# B&R Automation Studio project TD52 (part 8)

#### main.c
```c
/********************************************************************
 * COPYRIGHT -- Bernecker + Rainer Industrie-Elektronik Ges.m.b.H.
 ********************************************************************
 * Program: Sim3pCTR
 * File: main.c
 * Author: 105051472
 * Created: Thu Jan 10 08:03:20 2013
 ********************************************************************
 * Implementation of program Sim3pCTR
 ********************************************************************
 * Generated with B&R Automation Studio Target for Simulink V3.3
 * (ERT based)
 ********************************************************************/

#include <bur/plctypes.h>
#include "Sim3pCTR.h"
#include "rtwtypes.h"

BOOL bur_firsttime = TRUE;

/*  Defines */

/*  Data Types */

/**************************** GLOBAL DATA *************************************/
/*  Definitions */

/*  Declarations  */

/***************************** FILE SCOPE DATA ********************************/

/*************************** FUNCTIONS ****************************************/
#ifdef __cplusplus

unsigned long bur_heap_size = 65535;

#endif

void Sim3pCTR(struct Sim3pCTR* inst)
{
  switch (inst->ssMethodType)
  {
   case SS_INITIALIZE:
    /* call model initialize function */
    Sim3pCTR_initialize(inst);
    break;

   case SS_OUTPUT:
    /* call model step function */
    Sim3pCTR_step(inst);

    break;

   case SS_TERMINATE:
    /* call model terminate function */
    Sim3pCTR_terminate(inst);
    break;
  }
}

/*****************************************************************************
   Function block sample time: 0.01s
 *****************************************************************************/

/*****************************************************************************
   B&R Automation Studio Target for Simulink Version: V3.3.19 (13-Jun-2012)
 *****************************************************************************/

/*======================== TOOL VERSION INFORMATION ==========================*
 * MATLAB 7.12 (R2011a)09-Mar-2011                                            *
 * Simulink 7.7 (R2011a)09-Mar-2011                                           *
 * Simulink Coder 8.0 (R2011a)09-Mar-2011                                     *
 * Embedded Coder 6.0 (R2011a)09-Mar-2011                                     *
 * Stateflow 7.7 (R2011a)09-Mar-2011                                          *
 * Simulink Fixed Point 6.5 (R2011a)09-Mar-2011                               *
 *============================================================================*/

/*======================= LICENSE IN USE INFORMATION =========================*
 * matlab                                                                     *
 * matlab_coder                                                               *
 * real-time_workshop                                                         *
 * rtw_embedded_coder                                                         *
 * simulink                                                                   *
 * stateflow                                                                  *
 *============================================================================*/
```

#### lib_properties.txt
```
For manual assignment to hardware configuration please
add the following additional include directories:

\Logical\MATLAB_includes\R2011a\

And the following additional build options:

-lm -D MODEL=Sim3pCTR -D NUMST=1 -D NCSTATES=0 -D HAVESTDIO -D ONESTEPFCN=1 -D TERMFCN=1 -D MAT_FILE=0 -D MULTI_INSTANCE_CODE=0 -D INTEGER_CODE=0 -D MT=0 -D TID01EQ=0
```

### Library Logical/Libraries/ParaBase (IEC, version 4.13.0) - GE JEN engine parameter handling functions
Depends on: standard

#### ParaBase.typ - Exported data types
```iecst
TYPE
	MM2ParaBase_type : 	STRUCT
		bMySys_Run : BOOL; (*module is loaded and running on plc*)
		bMyParaSetupOk : BOOL; (*Modul confirms its OWN parameter to be OK with TRUE; USED FOR PERMANENT PART MODULES*)
		bMyParaMissing : BOOL; (*optional- Modul can indicate essentilal parameter errors with this bit to ParaBase (normaly the inversion of bMyParaSetupOk)  USE FOR FLEXIBLE PART MODULES*)
		bModuleMandatory : BOOL; (*optional- TRUE on this bit signals the ParaBase system, that engine operation is not allowed without this modules parameter OK (=change module to PERMANENT PART)*)
		iMyOwnModuleID : UDINT; (*Module ID code of a module with mandatory parameter missing*)
		iMyErrorInfo : UDINT; (*error status output of this single module*)
		iMyStateInfo : DINT; (*status output of this single module*)
		tMyProg_Vers : Revision_type; (*replacement for prog_vers, for this single module*)
		tClaimVisVersion : Revision_type; (*corequisite VISU version for this module*)
		iPermStatus : DINT; (*V4.06 - Debug Information: positive= checked perm items or files, negative= missed check info*)
		bPermSetupOk : BOOL; (*V4.06 - confirms (MODULE OWN) permanent data to be OK *)
	END_STRUCT;
	ParaBase2MM_type : 	STRUCT
		bParaSetupOk : BOOL; (*ALL mandatory modules signaled PARAMETER OK*)
		bSys_Run : BOOL; (*ALL modules are loaded and running on plc*)
		bDownloadDetected : BOOL; (*a program download was detected since last reboot, so paramter values may have been compromised and will not be stored*)
		bSaveParaAllowed : BOOL; (*no problems in parameter module, cyclic parameter saving is active*)
		bParaMissing : BOOL; (*Any mandatory module failed to confirm parameter OK status*)
		bParaWarning : BOOL; (*Any minor module failed to confirm parameter OK status*)
		iProg_Vers_Min : UDINT; (*replacement for prog_vers, LOWEST single module version*)
		iProg_Vers_Max : UDINT; (*info: max. prog_vers (to confirm newest update)*)
		iParaBaseExtensionAdress : UDINT; (*optional: prepared access point for unlisted modules*)
		iParaBaseExtensionCommand : UDINT; (*optional: prepared access point for unlisted modules*)
	END_STRUCT;
	ParaHandler_typ : 	STRUCT
		szMetaModuleName : STRING[2];
		bParaSetupOk : BOOL; (*confirms (OWN) parameter to be OK *)
		bThisParaCheckdOk : BOOL; (*confirms the actual selected parameter to be OK *)
		iParaOkChecked : UDINT; (*Debug Information: positive checked parameter lines*)
		tParaBase2MM : ParaBase2MM_type;
		tMM2ParaBase : MM2ParaBase_type;
	END_STRUCT;
	Revision_type : 	STRUCT
		xx : USINT; (*MAIN VERSION with HARD COMPATIBILE INTERFACE AREA*)
		yy : USINT; (*Versions with DOWNWARDS COMPATIBLE Interface*)
		zz : USINT; (*Version with internal changes only. NO INTERFACE CHANGES*)
		cc : USINT; (*cc=customized version*)
		aaaaa : UDINT; (*(optional) Build Number for exact revision reference OR for basisupdate versions*)
	END_STRUCT;
	ModuleInfo_type : 	STRUCT
		szMetaModuleName : STRING[2];
		bSysRun : BOOL; (*module states to be running*)
		bParaSetupOk : BOOL; (*confirms (MODULE OWN) parameter to be OK *)
		bModuleMandatory : BOOL; (*True= actualy NO engine operation without this module ok*)
		bModuleDownloadDetected : BOOL; (*True= download detected (module parameter relevant)*)
		iParaOkChecked : DINT; (*Debug Information: positive checked parameter lines V4,06 DINT replaces UDINT*)
		tRevision : Revision_type; (*xx.yy.cc.zz(.aaaaa) and BU*)
		tMM2ParaBase : MM2ParaBase_type; (*internal*)
	END_STRUCT;
	ParaCommand :
		(
		eSaveDataObjContentNow := 1,
		eRestoreDataObjContent := 2,
		eRestoreBackupDataObj := 3, (*Old! Do not use anymore, command is no longer supported*)
		eDeleteBackupDataObj := 4, (*Old! Do not use anymore, command is no longer supported*)
		eReadOutMETAContentNow := 5, (*fromV4.4*)
		eClearParaCommands := 8,
		eClearParaErrors := 9
		);
END_TYPE
```

#### ParaBase.fun - Exported functions and function blocks
```iecst
FUNCTION GetModuleCode : UDINT
	VAR_INPUT
		NameStringAdr : UDINT;
	END_VAR
	VAR CONSTANT
		ParaFUB_InAdr_Err : UDINT := 333333; (*error code: IN ADRESS IS MISSING*)
	END_VAR
END_FUNCTION

FUNCTION GetModuleName : UDINT (*FEHLT NOCH! (STRING[2] geht nicht?*)
	VAR_INPUT
	END_VAR
END_FUNCTION

FUNCTION DataCheckSumm : DINT
	VAR_INPUT
		tiEnableTime : DINT; (*FUNCTION ENABLE with >0; optional other values than 1 may be used  for error state returns*)
		iDataAdr : UDINT;
		iDataLenght : UDINT;
		iModuleCode : DINT; (*IN/OUT*)
	END_VAR
	VAR
		ulChecksum1 : UDINT;
		ulChecksum2 : UDINT;
		ulChecksum3 : UDINT;
		ulChkValue : UDINT;
		ulPMPointer : UDINT;
	END_VAR
	VAR CONSTANT
		ParaFUB_InAdr_Err : UDINT := 333333; (*error code: IN ADRESS IS MISSING*)
	END_VAR
END_FUNCTION

FUNCTION_BLOCK ParaCheckFUB (*FUB to check parameter value to be withhin defined range*)
	VAR_INPUT
		Enable : BOOL; (*Paracheck FUB enable*)
		Para : REAL; (*Adress of common modulecheck input object*)
		ParaRangeMIN : REAL; (*minimum value for parameter to check*)
		ParaRangeMAX : REAL; (*maximum value for parameter to check*)
		_ParaSysAdr : UDINT; (*internal*)
	END_VAR
	VAR_OUTPUT
		_ParaState : UDINT; (*debug info only; NORMALY USE OUTPUTS in  struct MM2ParaBase, e.g. .bMyParaSetupOk*)
	END_VAR
	VAR
		_tParaSys : REFERENCE TO ParaHandler_typ; (*internal (containing MM2ParaBase and ParaBase2MM Structures)*)
		_bAdressErr : BOOL; (*internal*)
	END_VAR
	VAR CONSTANT
		ParaFUB_SysAdr_Err : UDINT := 555555; (*error code: SYS ADRESS IS MISSING*)
		ParaFUB_SysRun_Err : UDINT := 888888; (*error code: necessary precondition to do ParaCheck is missing*)
		ParaFUB_Disabeled_Err : UDINT := 999999; (*error code: FUNCTION DISABELED *)
	END_VAR
END_FUNCTION_BLOCK
```

#### ParaBase.st
```iecst
(********************************************************************
 * COPYRIGHT -- INNIO Company
 ********************************************************************
 * Library: ParaBase
 * File: ParaBase.st
 * Author: zengerer
 * Created: August 01, 2012
 * V 0.12 2012-09-27 Ze,  Bugfix in bMyParaSetupOk
 * V 3.90 2013-03-22 Ze	  Type declarations
 * V 4.13 2023-11-20 Ze	  FUNCTION DataCheckSumm
 ********************************************************************

 *-------------------------------------------------------------------
 * Implementation of library ParaBase
 ********************************************************************)

(* Get module number coded from the 2-character module name *)
FUNCTION GetModuleCode
	IF NameStringAdr > 0 THEN
		(*get module code number from first 2 characters of module name*)
		memcpy(ADR(GetModuleCode), NameStringAdr,2); 		(*copy first 2 characters from clear text name to (ASCII) module code  *)
	ELSE
		GetModuleCode := ParaFUB_InAdr_Err;		(*Error message code*)

	END_IF

END_FUNCTION

(* Get 2-character module name from the module number coded  *)
FUNCTION GetModuleName		(* retired, never used *)

		GetModuleName := 33333;		(*Error message code*)

END_FUNCTION

(* Calculate Checksumm of Perm or Para Data Type  *)
FUNCTION DataCheckSumm
	IF tiEnableTime > 0 AND iDataAdr > 0 AND iDataLenght > 0 THEN	// AND iDataLenght < 500 THEN	(* Function inputs ok check *)

		ulChecksum1 := 0;
		ulChecksum2 := 0;
		ulChecksum3 := 0;

				FOR ulPMPointer := iDataAdr TO (iDataAdr + iDataLenght - SIZEOF(ulChkValue)) BY SIZEOF(ulChkValue) DO
					memcpy(ADR(ulChkValue), ulPMPointer, SIZEOF(ulChkValue));
					ulChecksum1 := ( ulChecksum1 XOR ulChkValue);
					ulChecksum2 := ( ulChecksum2 XOR ulChkValue) + ulChkValue  ;	(*test*)
					ulChecksum3 :=   ulChecksum3 XOR (ulChkValue * ulPMPointer);	(*test*)

				END_FOR;

				IF 	  iModuleCode = 2  THEN
					DataCheckSumm	:= ABS(ulChecksum2); 	(*allways output positive checksumm values*)
				ELSIF iModuleCode = 3 THEN
					DataCheckSumm	:= ABS(ulChecksum3);	(*allways output positive checksumm values*)
				ELSE
					DataCheckSumm	:= ABS(ulChecksum1);	(*allways output positive checksumm values*)
				END_IF
	ELSE
					DataCheckSumm :=  -ParaFUB_InAdr_Err;	(*Error message code, returned as negative value*)
	END_IF;

END_FUNCTION

(*-----------------------------------------------------------------------------*)

(* Check, if a parameter value is withhin the valid range *)
FUNCTION_BLOCK ParaCheckFUB
	IF Enable THEN
		(* Function Block state check *)
		IF _ParaSysAdr > 0 THEN
			_tParaSys ACCESS(_ParaSysAdr);		(*  Connect internal to global structure*)
			_bAdressErr	:= FALSE;
			_ParaState	:= 0;
		ELSE
			_bAdressErr	:= TRUE;
			_ParaState	:= ParaFUB_SysAdr_Err;		(*Error message code*)

		END_IF;

		IF _ParaState = 0 THEN 				(*Execute function ONLY WHEN ADRESSES ARE OK!*)
			(*-------------------------------------------------------------------------------*)
			IF _tParaSys.tParaBase2MM.bSys_Run THEN 				(* necessary precondition to do ParaCheck sucessfully*)

				(* parameter validity check *)
				_tParaSys.bThisParaCheckdOk :=        (Para >= ParaRangeMIN) AND (Para <= ParaRangeMAX);						(*checkpoint 'ParaOK' for only this instance of FUB*)

			ELSE
				_tParaSys.bThisParaCheckdOk := FALSE;
				_ParaState	:= ParaFUB_SysRun_Err;		(* necessary precondition to do ParaCheck sucessfully is missing*)
			END_IF

			_tParaSys.bParaSetupOk 					:= _tParaSys.bParaSetupOk 					AND _tParaSys.bThisParaCheckdOk;		(* checkpoint 'ParaOK' for ALL INSTANCES BEVORE AND INCLUDING THIS ONE !debug Info ONLY!*)
			_tParaSys.tMM2ParaBase.bMyParaSetupOk   := _tParaSys.tMM2ParaBase.bMyParaSetupOk  	AND _tParaSys.bThisParaCheckdOk;		(* checkpoint 'ParaOK' for ALL INSTANCES BEVORE AND INCLUDING THIS ONE !LIFE CONNECTED TAG!*)

			IF _tParaSys.tMM2ParaBase.bMyParaSetupOk	THEN _tParaSys.iParaOkChecked := _tParaSys.iParaOkChecked +1; END_IF			(* debug information *)

			(*--------------------------------------------------------------------------------*)
		END_IF

	ELSE
		_ParaState	:= ParaFUB_Disabeled_Err;				(* error code: FUNCTION DISABELED *)
	END_IF
END_FUNCTION_BLOCK
```

### Library Logical/Libraries/MBTCP (ANSIC, version 0.05.0) - ModBusTCP
Depends on: Runtime, standard, AsTCP, sys_lib, brsystem, asstring

#### MBTCP.fun - Exported functions and function blocks
```iecst
(********************************************************************
 * COPYRIGHT -- Bernecker + Rainer
 ********************************************************************
 * Library: MBTCP
 * File: MBTCP.fun
 * Author: B&R
 * Created: September 04, 2008
 ********************************************************************
 * Functions and function blocks of library MBTCP
 ********************************************************************)
(*Configures a Modbus over TCP slave (server) and provides a Modbus slave ID. fMBTSOpen() should be called in the INIT section of a task prior to fMBTSlave(). See also fMBTSClose() to close the slave in the EXIT section. This slave can then be read from, or written to, by fMBTMaster() or widely available Modbus over TCP programs.Hosts up to 127 Modbus units, each unit contains set of size-adjustable coils, discrete inputs, input registers, and holding registers. <a href="../MBTCP Slave/MBTCP Slave.html"> See Modbus Slave/Server for more information</a>*)

FUNCTION_BLOCK fMBTSOpen
	VAR_INPUT
		bEnable : BOOL; (*Enables the function block*)
		uiPort : UINT; (*TCP port number (default = 502) *)
		uiNbrCoils : UINT; (*Number of read-write binary coils*)
		uiNbrDiscreteInputs : UINT; (*Number of read-only binary discrete inputs *)
		uiNbrInputRegs : UINT; (*Number of read-only 16-bit input registers *)
		uiNbrHoldingRegs : UINT; (*Number of read-write 16-bit holding registers *)
		uiOffsetUnits : UINT; (*Offset of Modbus units. *)
		uiNbrUnits : UINT; (*Number of Modbus units. If external array are used this parameter has to be set to 1*)
		pbCoil : REFERENCE TO BOOL; (*Coil mapping, given as array of BOOL. Must be set to 0 if internal mapping is used*)
		pbDInp : REFERENCE TO BOOL; (*Discrete input mapping, given as array of BOOL. Must be set to 0 if internal mapping is used*)
		puiIReg : REFERENCE TO UINT; (*Input register mapping, given as array of UINT. Must be set to 0 if internal mapping is used*)
		puiHReg : REFERENCE TO UINT; (*Holding register mapping, given as array of UINT. Must be set to 0 if internal mapping is used*)
	END_VAR
	VAR_OUTPUT
		uiNbrAllocUnits : UINT; (*Number of actaully allocated units *)
		udiIdent : UDINT; (*Ident (pointer to memory area holding Modbus server structure)*)
		uiStatus : UINT; (*Status 0 for OK, otherwise <a href="../../Data types and constants/Constants.html"> Error Number </a>*)
	END_VAR
END_FUNCTION_BLOCK
(*Modbus/TCP slave (server) function. fMBTSlave() should be called in the CYCLIC section of a task after being configured by fMBTSOpen(). The server is closed by fMBTSClose(). This server can be read from or written to by fMBTMaster() or widely available Modbus over TCP programs. <a href="../MBTCP Slave/MBTCP Slave.html"> See Modbus Slave/Server for more information</a>*)

FUNCTION_BLOCK fMBTSlave
	VAR_INPUT
		bEnable : BOOL; (*Enables the function block*)
		udiIdent : UDINT; (*Ident, as provided in instfMBTSOpen.udiIdent *)
		tiRecvDelay : TIME; (*Time to wait before disconnecting a non-responding client (master)*)
	END_VAR
	VAR_OUTPUT
		usiClientNbr : UINT; (*How many clients (masters) are connected *)
		usiClientServed : USINT; (*Client (master) currently served *)
		tiRecvElapsed : TIME; (*Time spent waiting for response from Master *)
		usiUnit : USINT; (*Server unit read or written *)
		usiClientIP : STRING[18]; (*Client (master) IP address *)
		usiMBFuncCode : USINT; (*Modbus function code *)
		uiSentDataLen : UINT; (*Length of data sent *)
		szMsg : STRING[100]; (*Debug Message*)
		stTcpServerStatus : UINT; (*Status from the TCPServer function*)
		udiRecvCnt : UDINT; (*Counter receive data*)
		udiSendCnt : UDINT; (*Counter Send Data*)
		usiOpenRetries : USINT; (*Port open Retries*)
		CltInfo : ARRAY[0..4] OF tstclient_info; (*Client Info (IP-Adresse, Port, Ident)*)
		uiStep : UINT; (*Current step executed by the Slave's state machine*)
		uiStatus : UINT; (*Status 0 for OK, otherwise <a href="../../Data types and constants/Constants.html"> Error Number </a>*)
	END_VAR
END_FUNCTION_BLOCK
(*Terminates a Modbus/TCP slave (server) and releases allocated memory. fMBTSClose() should be called in the EXIT section of a task. See also fMBTSOpen() and fMBTSlave().*)

FUNCTION_BLOCK fMBTSClose
	VAR_INPUT
		bEnable : BOOL; (*Enables the function block*)
		udiIdent : UDINT; (*Ident, as provided in instfMBTSOpen.udiIdent *)
	END_VAR
	VAR_OUTPUT
		uiStatus : UINT; (*Status 0 for OK, otherwise <a href="../../Data types and constants/Constants.html"> Error Number </a>*)
	END_VAR
END_FUNCTION_BLOCK
(*Read/write individual values from/to coils and registers of given unit. The function code to use in member uiFcode of the passed structure is the same as for Modbus (0x01..0x06,0x0F,0x10,0x17) and two user defined functions (0x41,0x42). *)

FUNCTION_BLOCK fMBTSRW
	VAR_INPUT
		bEnable : BOOL; (*Enables the function block*)
		udiIdent : UDINT; (*Ident, as provided in instfMBTSOpen.udiIdent *)
		usiFCode : USINT; (*Modbus function code, see <a href="../../Data types and constants/Constants.html">constants</a>*)
		usiUnit : USINT; (*Unit to access*)
		uiReadAddr : UINT; (*Element in coil or register for read access*)
		uiReadQty : UINT; (*Quantity of coils/regs to read*)
		puiReadVal : REFERENCE TO UINT; (*Requested read value, pointer to UINT*)
		uiWriteAddr : UINT; (*Element in coil or register for write access*)
		uiWriteQty : UINT; (*Quantity of coils/regs to write*)
		puiWriteVal : REFERENCE TO UINT; (*Requested write value, pointer to UINT*)
	END_VAR
	VAR_OUTPUT
		uiStatus : UINT; (*Status 0 for OK, otherwise <a href="../../Data types and constants/Constants.html"> Error Number </a>*)
	END_VAR
END_FUNCTION_BLOCK
(*Initialize the slave's data units (coils and registers) with values. Coils and Discrete Inputs are initialized with 0, 1, 0... Input registers are filled with 1000, 1001, 1002... Holding registers are initialized with 0, 1, 2... *)

FUNCTION_BLOCK fMBTSFill
	VAR_INPUT
		bEnable : BOOL; (*Enables the function block*)
		udiIdent : UDINT; (*Ident, as provided in instfMBTSOpen.udiIdent *)
	END_VAR
	VAR_OUTPUT
		uiStatus : UINT; (*Status 0 for OK, otherwise <a href="../../Data types and constants/Constants.html"> Error Number </a>*)
	END_VAR
END_FUNCTION_BLOCK
(*Allocates memory and pre-configures Modbus TCP Master. fMBTMOpen() should be called in the INIT section of a task prior to fMBTMaster(). See also fMBTMClose() to close the master in the task's EXIT section. The master connects to the Modbus TCP slave available at the IP address provided by szSlvIPAddr. *)

FUNCTION_BLOCK fMBTMOpen
	VAR_INPUT
		bEnable : BOOL; (*Enables the function block*)
		szSlvIPAddr : STRING[18]; (*Slave's IP address *)
		uiPort : UINT; (*TCP port number (default = 502) *)
		uiRecvTimeout : UINT; (*Timeout to wait for answer from Slave prior to sending new request (default = 500 s) *)
	END_VAR
	VAR_OUTPUT
		udiIdent : UDINT; (*Ident (pointer to memory area holding Modbus Master structure)*)
		uiStatus : UINT; (*Status 0 for OK, otherwise <a href="../../Data types and constants/Constants.html"> Error Number </a>*)
	END_VAR
END_FUNCTION_BLOCK
(*Modbus/TCP master (client) function. fMBTMaster() should be called in the CYCLIC section of a task after being configured by fMBTMOpen(). The master is closed by fMBTMClose(). This master writes to or reads from a slave running fMBTSlave() or other widely available Modbus over TCP slave programs. *)

FUNCTION_BLOCK fMBTMaster
	VAR_INPUT
		bEnable : BOOL; (*Enables the function block*)
		udiIdent : UDINT; (*Ident, as provided in instfMBTMOpen.udiIdent *)
	END_VAR
	VAR_OUTPUT
		uiStep : UINT; (*Step executed by Master. Useful to monitor execution. *)
		uiTxID : UINT; (*Transaction ID *)
		usiMBFuncCode : USINT; (*Modbus function code *)
		szMsg : STRING[100]; (*Status from the TCPClient functions*)
		usiRxByteCnt : USINT; (*Number of bytes received from slave. See response byte count in Modbus protocol. *)
		uiStatus : UINT; (*Status 0 for OK, otherwise <a href="../../Data types and constants/Constants.html"> Error Number </a>*)
	END_VAR
END_FUNCTION_BLOCK
(*Terminates a Modbus/TCP master (client) and releases allocated memory. fMBTMClose() should be called in the EXIT section of a task. See also fMBTMOpen() and fMBTMaster(). *)

FUNCTION_BLOCK fMBTMClose
	VAR_INPUT
		bEnable : BOOL; (*Enables the function block*)
		udiIdent : UDINT; (*Ident, as provided in instfMBTMOpen.udiIdent *)
	END_VAR
	VAR_OUTPUT
		uiStatus : UINT; (*Status 0 for OK, otherwise <a href="../../Data types and constants/Constants.html"> Error Number </a>*)
	END_VAR
END_FUNCTION_BLOCK
(*Read/write individual values from/to coils and registers of given unit. The function code to use in member uiFcode of the passed structure is the same as for Modbus (0x01..0x06,0x0F,0x10,0x17).*)

FUNCTION_BLOCK fMBTMRW
	VAR_INPUT
		bEnable : BOOL; (*Enables the function block*)
		udiIdent : UDINT; (*Ident from fMBTMOpen*)
		usiFCode : USINT; (*Modbus function code, see <a href="../../Data types and constants/Constants.html">constants</a>*)
		usiUnit : USINT; (*Slave unit*)
		uiReadAddr : UINT; (*Element in coil or register for read access*)
		uiReadQty : UINT; (*Quantity of coils/regs to read*)
		puiReadVal : REFERENCE TO UINT; (*Requested read value, pointer to UINT*)
		uiWriteAddr : UINT; (*Element in coil or register for write access*)
		uiWriteQty : UINT; (*Quantity of coils/regs to write*)
		puiWriteVal : REFERENCE TO UINT; (*Requested write value, pointer to UINT*)
		bPoll : BOOL; (*Poll slave repeatedly (0 = single request)*)
		udiPollPeriod : UDINT; (*Polling period in ms*)
	END_VAR
	VAR_OUTPUT
		bRecvOK : BOOL; (*Confirms requested data was sent by slave*)
		uiStatus : UINT; (*Status 0 for OK, otherwise <a href="../../Data types and constants/Constants.html"> Error Number </a>*)
	END_VAR
END_FUNCTION_BLOCK
```

#### MBTCP.typ - Exported data types
```iecst
(********************************************************************
 * COPYRIGHT -- Bernecker + Rainer
 ********************************************************************
 * Library: MBTCP
 * File: MBTCP.typ
 * Author: B&R
 * Created: September 04, 2008
 ********************************************************************
 * Data types of library MBTCP
 ********************************************************************)
(*Client informationen*)

TYPE
	tstclient_info : 	STRUCT  (*Client information*)
		udiIdent : UDINT; (*Client Indentifier*)
		usiPort : USINT; (*Client Port*)
		szIp_addr : STRING[18]; (*Client IP- Adresse*)
		szMsg : STRING[100]; (*Client Message*)
	END_STRUCT;
END_TYPE
```

#### MBTCP.var - Exported constants
```iecst
(********************************************************************
 * COPYRIGHT -- Bernecker + Rainer
 ********************************************************************
 * Library: MBTCP
 * File: MBTCP.var
 * Author: B&R
 * Created: September 04, 2008
 ********************************************************************
 * Constants of library MBTCP <header> Error numbers below 50000 are from automation studio libraries and these are described in the automation studio help. </header>
 ********************************************************************)
VAR CONSTANT
	mbtERR_ILLEGAL_FUNCTION : UINT := 50001; (*Modbus function not implemented/non-existent *)
	mbtERR_DATA_ADDRESS : UINT := 50002; (*Address not available in coil or register *)
	mbtERR_IP_ADRESS : UINT := 50004; (*Wrong IP address passed to Master *)
	mbtERR_NBR_UNITS : UINT := 50005; (*Requested unit does not exist *)
	mbtERR_NULL_POINTER : UINT := 50006; (*Null pointer passed to function block *)
	mbtERR_MAX_CLIENT : UINT := 51001; (*Maximal amount of client is already connected *)
	mbtERR_NOT_CONNECTED : UINT := 51002; (*Half-open connection*)
	mbtERR_WR_ERROR_SOCKET : UINT := 51003; (*TCPServer socket error *)
	mbtERR_FATAL_ERROR : UINT := 51004; (*Fatal Error*)
	mbtERR_TIMEOUT : UINT := 51005; (*Modbus TCP timeout *)
	mbtERR_OPEN_RETRIES_IOC : UINT := 51006; (*Retried open port at the TCP IOControl *)
	mbtERR_OPEN_RETRIES_WR : UINT := 51007; (*Retried open port again at the TCPServer *)
	mbtERR_REQUEST_LEN_ZERO : UINT := 51008; (*The Server received a request with zero bytes *)
	mbtERR_MIN_FRAME_LEN : UINT := 51009; (*The Server received a request with a too short frame*)
	mbtERR_REQUEST_UNIT : UINT := 51010; (*Unit ID too high or low*)
	mbtERR_PROTOCOL_ID : UINT := 51011; (*Protocol ID != 0. Modbus Protocol ID must be 0 *)
	mbtERR_FCODE_ZERO : UINT := 51012; (*Function code is zero*)
	mbtERR_REQUEST : UINT := 51013; (*Request from client is wrong *)
	mbtERR_RESPONSE : UINT := 51014; (*Response from server is wrong *)
	mbtERR_MAX_NBR_COILS : UINT := 51015; (*Maximal number of coils is exceeded (2000) *)
	mbtERR_MAX_NBR_REGISTER : UINT := 51016; (*Maximal number of register is exceeded (127) *)
	mbtEVENT_OPEN_PORT : UINT := 52001; (*Opened new TCP Port *)
	mbtEVENT_ADD_CLIENT : UINT := 52002; (*Added new Client to the MBTCP Server*)
	mbtEVENT_IPADRESS_IDENT : UINT := 52003; (*Deploy ID with IP-adress. The ID is written in binary data at the logger*)
	mbtEVENT_CLOSE_CLIENT : UINT := 52004; (*Closed the Client connection *)
	mbtEVENT_CLOSE_PORT : UINT := 52005; (*Closed the Port*)
	MBT_READ_COILS : USINT := 1; (*Modbus function code: Read coils*)
	MBT_READ_DISCRETE_INPUTS : USINT := 2; (*Modbus function code: Read discrete inputs*)
	MBT_READ_HOLDING_REGISTERS : USINT := 3; (*Modbus function code: Read holding registers*)
	MBT_READ_INPUT_REGISTERS : USINT := 4; (*Modbus function code: Read input registers*)
	MBT_WRITE_SINGLE_COIL : USINT := 5; (*Modbus function code: Write single coil*)
	MBT_WRITE_SINGLE_REGISTER : USINT := 6; (*Modbus function code: Write single register (holding register)*)
	MBT_WRITE_MULTIPLE_COILS : USINT := 15; (*Modbus function code: Write multiple coils*)
	MBT_WRITE_MULTIPLE_REGISTERS : USINT := 16; (*Modbus function code: Write multiple registers (holding register)*)
	MBT_READ_WRITE_MULTIPLE_REGISTER : USINT := 23; (*Modbus function code: Read and write multiple registers*)
	BR_MBT_WRITE_DISCRETE_INPUTS : USINT := 65; (*User defined modbus function code: Write discrete inputs*)
	BR_MBT_WRITE_INPUT_REGISTERS : USINT := 66; (*User defined modbus function code: Write input register*)
END_VAR
```

#### fMBTSOpen.c
```c
/******************************************************************************
 * Copyright:    B&R Industrie-Automation AG
 *
 * Project:      Library MBTCP
 *
 * Target:       B&R-PCC
 *
 * AR-Version:   B 2.01
 *
 * AS-Version:   V 3.0.71.16.SP01
 *
 * Filename:     fMBTSOpen.c
 *
 * Function:     module-description
 *
 * Dependencies: description of all dependencies
 *
 ******************************************************************************
 * History:
 *
 * Version | Date        | Author       | Description
 * ----------------------------------------------------------------------------
 *    1.00 | 2008-sep-19 | H.Anderes    | creation
 *****************************************************************************/

/*****************************************************************************
 * includes
 *****************************************************************************/
/* ansi-c import */
/* system import */
/* user defined import */
#include "MBTCP.h"
#include "MBTSlave.h"

/*****************************************************************************
 * type definitions
 *****************************************************************************/

/*****************************************************************************
 * functions
 *****************************************************************************/
/*===========================================================================*/
void fMBTSOpen(struct fMBTSOpen* inst)
/*----------------------------------------------------------------------------
  Function:

  Configures a Modbus over TCP slave (server) and provides a Modbus
  slave ID. fMBTSOpen() should be called in the INIT section of a task
  prior to fMBTSlave(). See also fMBTSClose() to close the slave in
  the EXIT section. This slave can then be read from, or written to,
  by fMBTMaster() or widely available Modbus over TCP programs.

  History:

  Version | Date        | Author      | Description
  ----------------------------------------------------------------------------
  1.00    | 2008-sep-19 | H.Anderes   | creation
  1.01    | 2009-dez-03 | H.Anderes   | external structures
  ===========================================================================*/
{
  /* _LOCAL */
  UINT astatus    = 0;
  UINT i, u       = 0;
  BOOL extMapping = 0;
  /* _DYNAMIC */
  tstMBT_SVars *mbs;
  tstMBT_SData *pData;
  tCOIL *pCoils;
  tDINP *pDiscreteInputs;
  tIREG *pInputRegs;
  tHREG *pHoldingRegs;
  /*=========================================================================*/
  if (inst == NULL)
  {
    inst->uiStatus = mbtERR_NULL_POINTER;
    goto END;
  }
  if (inst->bEnable < TRUE)
  {
    inst->uiNbrAllocUnits = 0;
    inst->uiStatus = ERR_FUB_ENABLE_FALSE;
  }
  else
  {
    inst->uiStatus = ERR_FUB_BUSY;
    if (inst->uiPort < 1)
      inst->uiPort = MBT_SLAVE_PORT;

    if (inst->uiNbrUnits < 1)
      inst->uiNbrUnits = NUNITS_DEF;

   	if(inst->uiOffsetUnits > 255)
   	 { inst->uiStatus = mbtERR_NBR_UNITS; goto END; }

   	if((inst->uiOffsetUnits + inst->uiNbrUnits) > 256)
   	 { inst->uiStatus = mbtERR_NBR_UNITS; goto END; }

    astatus = TMP_alloc(sizeof(tstMBT_SVars), (void**)&mbs);
    if (astatus > 0) { inst->uiStatus = astatus; goto END; }
    memset(mbs, 0, sizeof(tstMBT_SVars));
    astatus = TMP_alloc(sizeof(tstMBT_SData), (void**)&pData);
    if (astatus > 0) { inst->uiStatus = astatus; goto END; }
    memset(pData, 0, sizeof(tstMBT_SData));
    mbs->pData = pData;

    /* allocate memory for coils and registers
     */
    mbs->pData->uiNbrUnits 		 = inst->uiNbrUnits;
    mbs->pData->uiOffsetUnits = inst->uiOffsetUnits;

    inst->uiNbrAllocUnits = 0;           /* num of allocated units */

   /* check if the mapping type is valid */
   if (   (inst->pbCoil  == NULL)
       && (inst->pbDInp  == NULL)
       && (inst->puiIReg == NULL)
       && (inst->puiHReg == NULL))
   {
     extMapping = FALSE;
   }
   else
   {
     extMapping = TRUE;
   }

    for (u = inst->uiOffsetUnits; u < (inst->uiNbrUnits + inst->uiOffsetUnits); u++)
    {
      if (    (inst->pbCoil == NULL)
           && (inst->uiNbrCoils > 0))
      {
        astatus = TMP_alloc(inst->uiNbrCoils * sizeof(tCOIL),
                            (void **) &pCoils);
        if (astatus > 0) { inst->uiStatus = astatus; goto END; }
        memset((tCOIL *) pCoils, 0,
               inst->uiNbrCoils * sizeof(tCOIL));
        mbs->pData->stUnit[u].pCoils = (tCOIL *) pCoils;
        mbs->pData->stUnit[u].uiNbrCoils = inst->uiNbrCoils;
      }
      else if (    (inst->pbCoil != NULL)
                && (inst->uiNbrCoils > 0))
      {
        mbs->pData->stUnit[u].pCoils       = (tCOIL *) inst->pbCoil;
        mbs->pData->stUnit[u].uiNbrCoils   = inst->uiNbrCoils;
        mbs->pData->stUnit[0].bCoilsExtern = TRUE;
      }

      if (    (inst->pbDInp == NULL)
           && (inst->uiNbrDiscreteInputs > 0))
      {
        astatus = TMP_alloc(inst->uiNbrDiscreteInputs * sizeof(tDINP),
                            (void **) &pDiscreteInputs);
        if (astatus > 0) { inst->uiStatus = astatus; goto END; }
        memset((tDINP *) pDiscreteInputs, 0,
               inst->uiNbrDiscreteInputs * sizeof(tDINP));
        mbs->pData->stUnit[u].pDiscreteInputs = (tDINP *) pDiscreteInputs;
        mbs->pData->stUnit[u].uiNbrDiscreteInputs = inst->uiNbrDiscreteInputs;
      }
      else
      {
        mbs->pData->stUnit[u].pDiscreteInputs        = (tDINP *)  inst->pbDInp;
        mbs->pData->stUnit[u].uiNbrDiscreteInputs    = inst->uiNbrDiscreteInputs;
        mbs->pData->stUnit[0].bDiscreteInputsExtern  = TRUE;
      }

      if (    (inst->puiIReg == NULL)
           && (inst->uiNbrInputRegs > 0))
      {
        astatus = TMP_alloc(inst->uiNbrInputRegs * sizeof(tIREG),
                            (void **) &pInputRegs);
        if (astatus > 0) { inst->uiStatus = astatus; goto END; }
        memset((tIREG *) pInputRegs, 0,
               inst->uiNbrInputRegs * sizeof(tIREG));
        mbs->pData->stUnit[u].pInputRegs = (tIREG *) pInputRegs;
        mbs->pData->stUnit[u].uiNbrInputRegs = inst->uiNbrInputRegs;
      }
      else
      {
        mbs->pData->stUnit[u].pInputRegs        = (tIREG *)  inst->puiIReg;
        mbs->pData->stUnit[u].uiNbrInputRegs    = inst->uiNbrInputRegs;
        mbs->pData->stUnit[0].bInputRegsExtern  = TRUE;
      }

      if (    (inst->puiHReg == NULL)
           && (inst->uiNbrHoldingRegs > 0))
      {
        astatus = TMP_alloc(inst->uiNbrHoldingRegs * sizeof(tHREG),
                            (void **) &pHoldingRegs);
        if (astatus > 0) { inst->uiStatus = astatus; goto END; }
        memset((tHREG *) pHoldingRegs, 0,
               inst->uiNbrHoldingRegs * sizeof(tHREG));
        mbs->pData->stUnit[u].pHoldingRegs = (tHREG *) pHoldingRegs;
        mbs->pData->stUnit[u].uiNbrHoldingRegs = inst->uiNbrHoldingRegs;
      }
      else
      {
        mbs->pData->stUnit[u].pHoldingRegs        = (tHREG *) inst->puiHReg;
        mbs->pData->stUnit[u].uiNbrHoldingRegs    = inst->uiNbrHoldingRegs;
        mbs->pData->stUnit[0].bHoldingRegsExtern  = TRUE;
      }

      inst->uiNbrAllocUnits = inst->uiNbrAllocUnits + 1;

      /* if external mapping is used, only one mapping is allowed */
      if (extMapping == TRUE)
      {
        break;
      }
    }

    mbs->uiPort       = inst->uiPort;
    mbs->uiStep       = INIT;
    mbs->uiReturnStep = INIT;
    mbs->usiCltNr = 0;

    for (i = 0; i < MAX_CLIENT; i++)
    {
      mbs->TOFRecv[i].IN = TRUE;                       /* reset timer */
      TOF(&(mbs->TOFRecv[i]));
    }

    inst->udiIdent = (UDINT) mbs;
    if (inst->uiStatus == ERR_FUB_BUSY)                 /* alloc OK */
    {
      inst->uiNbrAllocUnits = inst->uiNbrAllocUnits;
      inst->uiStatus = ERR_OK;
    }
  }
END: ; /* do nothing */
  /*=========================================================================*/
} /* fMBTSOpen */

/*****************************************************************************
 * END OF CODE
 *****************************************************************************/
/*
  Local Variables:
  c-file-style: bsd
  c-basic-offset: 2
  comment-column: 45
  End:
*/
```

#### fMBTSlave.c
```c
/*****************************************************************************
 * Copyright:    B&R Industrie-Automation AG
 *
 * Project:      Library MBTCP
 *
 * Target:       B&R-PCC
 *
 * AR-Version:   B 2.01
 *
 * AS-Version:   V 3.0.71.16.SP01
 *
 * Filename:     fMBTSlave.c
 *
 * Function:     module-description
 *
 * Dependencies: description of all dependencies
 *
 *****************************************************************************
 * History:
 *
 * Version | Date        | Author      | Description
 * --------------------------------------------------------------------------
 *    1.00 | 2008-sep-19 | H.Anderes   | creation
 *****************************************************************************/

/*****************************************************************************
 * includes
 *****************************************************************************/
/* ansi-c import */
/* system import */
/* user defined import */
#include "MBTCP.h"
#include "MBTSlave.h"

/*****************************************************************************
 * type definitions
 *****************************************************************************/

/*****************************************************************************
 * functions
 *****************************************************************************/
/*===========================================================================*/
void fMBTSlave(struct fMBTSlave* inst)
/*----------------------------------------------------------------------------
  Function:

  Modbus/TCP slave (server) function. fMBTSlave() should be called in
  the CYCLIC section of a task after being configured by
  fMBTSOpen(). The server is closed by fMBTSClose(). This server can
  be read from or written to by fMBTMaster() or widely available
  Modbus over TCP programs.

  History:

  Version | Date        | Author      | Description
  --------------------------------------------------------------------------
  1.00    | 2008-sep-19 | H.Anderes   | creation
  2.00    | 2010-okt-04 | H.Anderes   | refactory
  ===========================================================================*/
{
  /* _LOCAL */
  /* _DYNAMIC */
  tstMBT_SVars* mbs;
  UINT i;
  /*=========================================================================*/
  /* check if nil pointer */
  if (inst == NULL || inst->udiIdent == 0)
  {
    inst->uiStatus = mbtERR_NULL_POINTER;
    goto END;
  }
  mbs = (tstMBT_SVars *) inst->udiIdent;

  if (inst->bEnable < TRUE)
  {
    inst->uiStatus = ERR_FUB_ENABLE_FALSE;
  }
  else
  {
    mbs->bEnable = inst->bEnable;
    for(i = 0; i < MAX_CLIENT; i++)          /* timeout setting */
    {
      if (inst->tiRecvDelay > 0)
      {
        mbs->TOFRecv[i].PT = inst->tiRecvDelay;
      }
      else
      {
        mbs->TOFRecv[i].PT = TIMEOUT_MS;
      }
    }
    /* call  fMBTSStates() */
    fMBTSStates(mbs);

    /* copy internal to the fub interface */
    inst->uiStatus          = mbs->uiStatus;
    inst->uiStep            = mbs->uiStep;
    inst->usiClientNbr      = mbs->usiCltNr;
    inst->usiClientServed   = mbs->usiCltServed;
    inst->tiRecvElapsed     = mbs->TOFRecv[mbs->usiCltServed].ET; /* timeout */
    strcpy(inst->usiClientIP, mbs->cltInfo[mbs->usiCltServed].szIp_addr);
    inst->usiUnit           = mbs->stRecvBuf[mbs->usiCltServed].byte[6];
    inst->usiMBFuncCode     = mbs->stRecvBuf[mbs->usiCltServed].byte[7];
   	strcpy(inst->szMsg, mbs->szMsg);
   	inst->stTcpServerStatus = mbs->stTcpServer.status;
   	inst->usiOpenRetries    = mbs->usiOpenRetries;
   	inst->udiRecvCnt        = mbs->udiRecvCnt;
   	inst->udiSendCnt        = mbs->udiSendCnt;
    /* get client information for debugging */
    for(i = 0; i < MAX_CLIENT; i++)
    {
    	 inst->CltInfo[i].udiIdent = mbs->cltInfo[i].udiIdent;
    	 inst->CltInfo[i].usiPort = mbs->cltInfo[i].usiPort;
      strcpy(inst->CltInfo[i].szIp_addr,mbs->cltInfo[i].szIp_addr);
      strcpy(inst->CltInfo[i].szMsg,mbs->cltInfo[i].szMsg);
    }
  }

END: ; /* do nothing */
  /*=========================================================================*/
} /* fMBTSlave */

/*****************************************************************************
 * END OF CODE
 *****************************************************************************/
/*
  Local Variables:
  c-file-style: bsd
  c-basic-offset: 2
  comment-column: 45
  End:
*/
```

#### fMBTSClose.c
```c
/*****************************************************************************
 * Copyright:    B&R Industrie-Automation AG
 *
 * Project:      Library MBTCP
 *
 * Target:       B&R-PCC
 *
 * AR-Version:   B 2.01
 *
 * AS-Version:   V 3.0.71.16.SP01
 *
 * Filename:     fMBTSClose.c
 *
 * Function:     module-description
 *
 * Dependencies: description of all dependencies
 *
 *****************************************************************************
 * History:
 *
 * Version | Date        | Author      | Description
 * ---------------------------------------------------------------------------
 *    1.00 | 2008-sep-19 | H.Anderes   | creation
 *****************************************************************************/

/*****************************************************************************
 * includes
 *****************************************************************************/
/* ansi-c import */
/* system import */
/* user defined import */
#include "MBTCP.h"
#include "MBTSlave.h"

/*****************************************************************************
 * type definitions
 *****************************************************************************/

/*****************************************************************************
 * functions
 *****************************************************************************/
/*===========================================================================*/
void fMBTSClose(struct fMBTSClose* inst)
/*----------------------------------------------------------------------------
  Function:

  Terminates a Modbus/TCP slave (server) and releases allocated
  memory.  fMBTSClose() should be called in the EXIT section of a
  task. See also fMBTSOpen() and fMBTSlave().

  History:

  Version | Date        | Author      | Description
  ----------------------------------------------------------------------------
     1.00 | 2008-sep-19 | H.Anderes    | creation
     5.00 | 2021-may-07 | W.Froehlich  | set correct FUB state fMBTSClose.uiStatus from ERR_FUB_BUSY to ERR_OK
  ===========================================================================*/
{
  /* _LOCAL */
  UINT u, c, fstatus = 0;
  USINT usiClientNr;
  /* _DYNAMIC */
  tstMBT_SVars* mbs;
  /*=========================================================================*/
  /* check if nil pointer */
  if (inst == NULL || inst->udiIdent == 0)
  {
    inst->uiStatus = mbtERR_NULL_POINTER;
	   goto END;
  }
  mbs = (tstMBT_SVars *)inst->udiIdent;

  if (inst->bEnable < TRUE)
  {
    inst->uiStatus = ERR_FUB_ENABLE_FALSE;
  }
  else
  {
		/* set correct FUB state fMBTSClose.uiStatus from ERR_FUB_BUSY to ERR_OK */
    inst->uiStatus = ERR_OK;

    /* disconnect all clients and close slave's port */
    mbs->uiStep = CLOSE_SLAVE;
    usiClientNr = mbs->usiCltNr;
    /* call fMBTSStates() */
    fMBTSStates(mbs);  /* internal main state machine */
    c = 0;
    while (    (mbs->bClosing > 0)
            && (c < MAX_CLOSE_LOOPS))
    {
      fMBTSStates(mbs);
      c++;
    }

    for (u = 0; u < mbs->pData->uiNbrUnits; u++)
    {
      if (mbs->pData->stUnit[0].bCoilsExtern == FALSE)
      {
        fstatus = TMP_free(mbs->pData->stUnit[u].uiNbrCoils * sizeof(tCOIL),
                             (void**)(mbs->pData->stUnit[u].pCoils));
        if (fstatus > 0)
        {
          inst->uiStatus = fstatus;
          ERRxwarning(fstatus, 0,
                      (STRING*)"fMBTSClose: failed to TMP_free pCoils");
          goto END;  /* EXIT_FAILURE; */
        }
      }

      if (mbs->pData->stUnit[0].bDiscreteInputsExtern == FALSE)
      {
        fstatus =
          TMP_free(mbs->pData->stUnit[u].uiNbrDiscreteInputs * sizeof(tDINP),
                   (void**)(mbs->pData->stUnit[u].pDiscreteInputs));
        if (fstatus > 0)
        {
          inst->uiStatus = fstatus;
          ERRxwarning(fstatus, 0,
                      (STRING*)"fMBTSClose: failed to TMP_free pDiscreteInputs");
          goto END;  /* EXIT_FAILURE; */
        }
      }

      if (mbs->pData->stUnit[0].bInputRegsExtern == FALSE)
      {
        fstatus = TMP_free(mbs->pData->stUnit[u].uiNbrInputRegs * sizeof(tIREG),
                           (void**)(mbs->pData->stUnit[u].pInputRegs));
        if (fstatus > 0)
        {
          inst->uiStatus = fstatus;
          ERRxwarning(fstatus, 0,
                      (STRING*)"fMBTSClose: failed to TMP_free pInputRegs");
          goto END;  /* EXIT_FAILURE; */
        }
      }

      if (mbs->pData->stUnit[0].bHoldingRegsExtern == FALSE)
      {
        fstatus = TMP_free(mbs->pData->stUnit[u].uiNbrHoldingRegs * sizeof(tHREG),
                           (void**)(mbs->pData->stUnit[u].pHoldingRegs));
        if (fstatus > 0)
        {
          inst->uiStatus = fstatus;
          ERRxwarning(fstatus, 0,
                      (STRING*)"fMBTSClose: failed to TMP_free pHoldingRegs");
          goto END;  /* EXIT_FAILURE; */
        }
      }
    }

    fstatus = TMP_free(sizeof(tstMBT_SData), (void**)mbs->pData);
    if (fstatus > 0)
    {
      inst->uiStatus = fstatus;
      ERRxwarning(fstatus, 0,
                  (STRING*)"fMBTSClose: failed to TMP_free pData");
        goto END;  /* EXIT_FAILURE; */
    }
    fstatus = TMP_free(sizeof(tstMBT_SVars), (void**)mbs);
		inst->udiIdent = 0;
    if (fstatus > 0)
    {
      inst->uiStatus = fstatus;
      ERRxwarning(fstatus, 0, (STRING*)"fMBTSClose: failed to TMP_free mbs");
      goto END;  /* EXIT_FAILURE; */
    }
  }
  END: ; /* do nothing */
  /*=========================================================================*/
  } /* fMBTSClose */

/*****************************************************************************
 * END OF CODE
 *****************************************************************************/
/*
Local Variables:
c-file-style: bsd
c-basic-offset: 2
comment-column: 45
End:
 */
```

#### fMBTSRW.c
```c
/*****************************************************************************
 * Copyright:    B&R Industrie-Automation AG
 *
 * Project:      Library MBTCP
 *
 * Target:       B&R-PCC
 *
 * AR-Version:   B 2.01
 *
 * AS-Version:   V 3.0.71.16.SP01
 *
 * Filename:     fMBTSRW.c
 *
 * Function:     module-description
 *
 * Dependencies: description of all dependencies
 *
 *****************************************************************************
 * History:
 *
 * Version | Date        | Author      | Description
 * --------------------------------------------------------------------------
 *    1.00 | 2008-sep-25 | H.Anderes    | creation
 *****************************************************************************/

/*****************************************************************************
 * includes
 *****************************************************************************/
/* ansi-c import */
/* system import */
/* user defined import */
#include "MBTCP.h"
#include "MBTSlave.h"

/*****************************************************************************
 * type definitions
 *****************************************************************************/

/*****************************************************************************
 * functions
 *****************************************************************************/
/*===========================================================================*/
void fMBTSRW(struct fMBTSRW* inst)
/*---------------------------------------------------------------------------
  Function:
  <header>
  <p>
   Read/write individual values from/to coils and registers of given unit.
   The function code to use in member uiFcode of the passed structure is the
   same as for Modbus (0x01..0x06) and two user defined functions (0x41,0x42).
   See Modbus function codes.

  History:

  Version | Date        | Author      | Description
  --------------------------------------------------------------------------
  1.00 | 2008-sep-19 | H.Anderes    | creation
  1.01 | 2009-mar-03 | H.Anderes   | implementation FC15, FC16
  1.01 | 2009-dez-09 | H.Anderes   | implementation FC23, change FUB interface
  ===========================================================================*/
{
  /* _LOCAL */
  UINT u, i;
  UINT coil;
  UINT hreg;
  UINT ireg;
  /* _DYNAMIC */
  tstMBT_SVars* mbs;
  tCOIL* pCoilVal;
  tDINP* pDInpVal;
  tIREG* pIRegVal;
  tHREG* pHRegVal;
  /*=========================================================================*/
  /* check if nil pointer */
  if (inst == NULL || inst->udiIdent == 0)
  {
    inst->uiStatus = mbtERR_NULL_POINTER;
	   goto END;
  }
  mbs = (tstMBT_SVars *) inst->udiIdent;

  if (inst->bEnable < TRUE)
  {
    inst->uiStatus = ERR_FUB_ENABLE_FALSE;
  }
  else
  {
    inst->uiStatus = ERR_FUB_BUSY;

    u = inst->usiUnit;
    if (    (u >= mbs->pData->uiNbrUnits + mbs->pData->uiOffsetUnits)
         || (u < mbs->pData->uiOffsetUnits))
      { inst->uiStatus = mbtERR_NBR_UNITS; goto END; }

    switch(inst->usiFCode)
    {
    /*------------------------------------------------------------------------
      READ: read coils
    -------------------------------------------------------------------------*/
    case MBT_READ_COILS:                     /* 0x01 */
      if (inst->puiReadVal == NULL)
        { inst->uiStatus = mbtERR_DATA_ADDRESS; goto END; }
      pCoilVal = (tCOIL*) inst->puiReadVal;
      i = inst->uiReadAddr;
      if (i > mbs->pData->stUnit[u].uiNbrCoils)
        { inst->uiStatus = mbtERR_DATA_ADDRESS; goto END; }
      if (    (inst->uiReadQty > 0)
           && (inst->uiReadQty <= (*(mbs->pData)).stUnit[u].uiNbrCoils))
      {
        if (    (inst->uiReadAddr + inst->uiReadQty)
             <= (*(mbs->pData)).stUnit[u].uiNbrCoils)
        {
          for (i = 0; i < inst->uiReadQty; i++)
          {
            coil = inst->uiReadAddr + i;
            if(((*(mbs->pData)).stUnit[u].pCoils[(i)] & (USINT)(0x01)))
              pCoilVal[(i)*2 + BYTE_OFFSET]  = (tCOIL) 1;
            else
              pCoilVal[(i)*2 + BYTE_OFFSET]  = (tCOIL) 0;
           }
        }
      }
      break;
	   /*-------------------------------------------------------------------------
      READ: read discrete inputs
    --------------------------------------------------------------------------*/
    case MBT_READ_DISCRETE_INPUTS:           /* 0x02 */
     if (inst->puiReadVal == NULL)
        { inst->uiStatus = mbtERR_DATA_ADDRESS; goto END; }
      pDInpVal = (tDINP*) inst->puiReadVal;
      i = inst->uiReadAddr;
      if (i > mbs->pData->stUnit[u].uiNbrDiscreteInputs)
        { inst->uiStatus = mbtERR_DATA_ADDRESS; goto END; }
      if (   (inst->uiReadQty > 0)
          && (inst->uiReadQty <= (*(mbs->pData)).stUnit[u].uiNbrDiscreteInputs))
      {
        if (    (inst->uiReadAddr + inst->uiReadQty)
             <= (*(mbs->pData)).stUnit[u].uiNbrDiscreteInputs)
        {
          for (i = 0; i < inst->uiReadQty; i++)
          {
            coil = inst->uiReadAddr + i;
            if(((*(mbs->pData)).stUnit[u].pDiscreteInputs[(i)] & (USINT)(0x01)))
              pDInpVal[(i)*2 + BYTE_OFFSET]  = (tCOIL) 1;
            else
              pDInpVal[(i)*2 + BYTE_OFFSET]  = (tCOIL) 0;
           }
        }
      }
      break;
	   /*--------------------------------------------------------------------------
      READ: read discrete inputs
    ---------------------------------------------------------------------------*/
    case MBT_READ_HOLDING_REGISTERS:         /* 0x03 */
      if (inst->puiReadVal == NULL)
        { inst->uiStatus = mbtERR_DATA_ADDRESS; goto END; }
      pHRegVal = (tHREG*) inst->puiReadVal;
      i = inst->uiReadAddr;
      if (i > mbs->pData->stUnit[u].uiNbrHoldingRegs)
        { inst->uiStatus = mbtERR_DATA_ADDRESS; goto END; }
      if (    (inst->uiReadQty > 0)
           && (inst->uiReadQty <= (*(mbs->pData)).stUnit[u].uiNbrHoldingRegs))
      {
        if (    (inst->uiReadAddr + inst->uiReadQty)
             <= (*(mbs->pData)).stUnit[u].uiNbrHoldingRegs)
        {
          for (i = 0; i < inst->uiReadQty; i++)
          {
            hreg = inst->uiReadAddr + i;
            pHRegVal[(i)] = mbs->pData->stUnit[u].pHoldingRegs[hreg];
          }
        }
      }
      break;
	   /*--------------------------------------------------------------------------
      READ: read input registers
    ---------------------------------------------------------------------------*/
    case MBT_READ_INPUT_REGISTERS:           /* 0x04 */
      if (inst->puiReadVal == NULL)
        { inst->uiStatus = mbtERR_DATA_ADDRESS; goto END; }
      pIRegVal = (tIREG*) inst->puiReadVal;
      i = inst->uiReadAddr;
      if (i > mbs->pData->stUnit[u].uiNbrInputRegs)
        { inst->uiStatus = mbtERR_DATA_ADDRESS; goto END; }
      if (    (inst->uiReadQty > 0)
           && (inst->uiReadQty <= (*(mbs->pData)).stUnit[u].uiNbrInputRegs))
        {
          if (    (inst->uiReadAddr + inst->uiReadQty)
               <= (*(mbs->pData)).stUnit[u].uiNbrInputRegs)
          {
            for (i = 0; i < inst->uiReadQty; i++)
            {
              ireg = inst->uiReadAddr + i;
              pIRegVal[(i)] = mbs->pData->stUnit[u].pInputRegs[ireg];
            }
          }
        }
      break;
	   /*--------------------------------------------------------------------------
      WRITE: write single coil
    ---------------------------------------------------------------------------*/
    case MBT_WRITE_SINGLE_COIL:              /* 0x05 */
     if (inst->puiWriteVal == NULL)
        { inst->uiStatus = mbtERR_DATA_ADDRESS; goto END; }
      pCoilVal = (tCOIL*) inst->puiWriteVal+BYTE_OFFSET;
      i = inst->uiWriteAddr;
      if (i > mbs->pData->stUnit[u].uiNbrCoils)
        { inst->uiStatus = mbtERR_DATA_ADDRESS; goto END; }
      mbs->pData->stUnit[u].pCoils[i] = *pCoilVal;
      break;
	   /*--------------------------------------------------------------------------
      WRITE: write single register
    ---------------------------------------------------------------------------*/
    case MBT_WRITE_SINGLE_REGISTER:          /* 0x06 */
      if (inst->puiWriteVal == NULL)
        { inst->uiStatus = mbtERR_DATA_ADDRESS; goto END; }
      pHRegVal = (tHREG*) inst->puiWriteVal;
      i = inst->uiWriteAddr;
   	  if (i > mbs->pData->stUnit[u].uiNbrHoldingRegs)
           { inst->uiStatus = mbtERR_DATA_ADDRESS; goto END; }
       mbs->pData->stUnit[u].pHoldingRegs[i] = *pHRegVal;
 	    break;
	   /*--------------------------------------------------------------------------
      WRITE: write discrete inputs
    ---------------------------------------------------------------------------*/
 	  case BR_MBT_WRITE_DISCRETE_INPUTS:       /* 0x41 */
      if (inst->puiWriteVal == NULL)
        { inst->uiStatus = mbtERR_DATA_ADDRESS; goto END; }
      pDInpVal = (tDINP*) inst->puiWriteVal;
      i = inst->uiWriteAddr;
   	  if (i > mbs->pData->stUnit[u].uiNbrDiscreteInputs)
           { inst->uiStatus = mbtERR_DATA_ADDRESS; goto END; }
      if (    (inst->uiWriteQty > 0)
            && (inst->uiWriteQty <= (*(mbs->pData)).stUnit[u].uiNbrDiscreteInputs))
      {
        if (    (inst->uiWriteAddr + inst->uiWriteQty)
             <= (*(mbs->pData)).stUnit[u].uiNbrDiscreteInputs)
        {
           for (i = 0; i < inst->uiWriteQty; i++)
           {
             coil = inst->uiWriteAddr + i;

             if((pDInpVal[(i*2)+ BYTE_OFFSET] & (USINT)(0x01)))
                 (*(mbs->pData)).stUnit[u].pDiscreteInputs[coil] = (tCOIL) 1;
             else
                 (*(mbs->pData)).stUnit[u].pDiscreteInputs[coil] = (tCOIL) 0;
            }
        }
      }
 	    break;
	  	/*--------------------------------------------------------------------------
      WRITE: write input register
    ---------------------------------------------------------------------------*/
 	  case BR_MBT_WRITE_INPUT_REGISTERS:        /* 0x42 */
      if (inst->puiWriteVal == NULL)
        { inst->uiStatus = mbtERR_DATA_ADDRESS; goto END; }
      pIRegVal = (tIREG*) inst->puiWriteVal;
      i = inst->uiWriteAddr;
   	  if (i > mbs->pData->stUnit[u].uiNbrInputRegs)
           { inst->uiStatus = mbtERR_DATA_ADDRESS; goto END; }
      if (   (inst->uiWriteQty > 0)
          && (inst->uiWriteQty <= (*(mbs->pData)).stUnit[u].uiNbrInputRegs))
       {
        if (   (inst->uiWriteAddr + inst->uiWriteQty)
            <= (*(mbs->pData)).stUnit[u].uiNbrInputRegs)
        {
          for (i = 0; i < inst->uiWriteQty; i++)
          {
            ireg = inst->uiWriteAddr + i;
            (*(mbs->pData)).stUnit[u].pInputRegs[ireg] = pIRegVal[(i)];
          }
        }
      }
      break;
	  	/*-------------------------------------------------------------------------
      WRITE: write multiple coils
    --------------------------------------------------------------------------*/
    case MBT_WRITE_MULTIPLE_COILS:           /* 0x0F */
      if (inst->puiWriteVal == NULL)
        { inst->uiStatus = mbtERR_DATA_ADDRESS; goto END; }
      pCoilVal = (tCOIL*) inst->puiWriteVal;
      i = inst->uiWriteAddr;
      if (i > mbs->pData->stUnit[u].uiNbrCoils)
        { inst->uiStatus = mbtERR_DATA_ADDRESS; goto END; }
    		if (    (inst->uiWriteQty > 0)
    	      && (inst->uiWriteQty <= (*(mbs->pData)).stUnit[u].uiNbrCoils))
    		{
  	    	if (    (inst->uiWriteAddr + inst->uiWriteQty)
  	         	<= (*(mbs->pData)).stUnit[u].uiNbrCoils)
  	    	{
  	        for (i = 0; i < inst->uiWriteQty; i++)
  	      		{
  	          coil = inst->uiWriteAddr + i;

  						     if((pCoilVal[(i)*2+BYTE_OFFSET]& (USINT)(0x01)))
  		          			(*(mbs->pData)).stUnit[u].pCoils[coil] = (tCOIL) 1;
  		        	else
  		          			(*(mbs->pData)).stUnit[u].pCoils[coil] = (tCOIL) 0;
  			       }
  		     }
    		}
		   break;
    /*--------------------------------------------------------------------------
      WRITE: write multiple register
    ---------------------------------------------------------------------------*/
    case MBT_WRITE_MULTIPLE_REGISTERS:       /* 0x10 */
      if (inst->puiWriteVal == NULL)
        { inst->uiStatus = mbtERR_DATA_ADDRESS; goto END; }
      pHRegVal = (tHREG*) inst->puiWriteVal;
      i = inst->uiWriteAddr;
      if (i > mbs->pData->stUnit[u].uiNbrHoldingRegs)
        { inst->uiStatus = mbtERR_DATA_ADDRESS; goto END; }
    		if (    (inst->uiWriteQty > 0)
          	&& (inst->uiWriteQty <= (*(mbs->pData)).stUnit[u].uiNbrHoldingRegs))
      		{
    		   if (   (inst->uiWriteAddr + inst->uiWriteQty)
    		       <= (*(mbs->pData)).stUnit[u].uiNbrHoldingRegs)
    		   {
    		     for (i = 0; i < inst->uiWriteQty; i++)
    		     {
    				     hreg = inst->uiWriteAddr + i;
    		       (*(mbs->pData)).stUnit[u].pHoldingRegs[hreg] = pHRegVal[(i)];
    		     }
    		   }
    		}
	     break;
    /*--------------------------------------------------------------------------
      WRITE: read and write multiple register
    ---------------------------------------------------------------------------*/
    case READ_WRITE_MULTIPLE_REGISTERS:
      /*****************write multiple register ***************/
      if (inst->puiWriteVal == NULL)
        { inst->uiStatus = mbtERR_DATA_ADDRESS; goto END; }
      pHRegVal = (tHREG*) inst->puiWriteVal;
      i = inst->uiWriteAddr;
      if (i > mbs->pData->stUnit[u].uiNbrHoldingRegs)
        { inst->uiStatus = mbtERR_DATA_ADDRESS; goto END; }
      if (    (inst->uiWriteQty > 0)
           && (inst->uiWriteQty <= (*(mbs->pData)).stUnit[u].uiNbrHoldingRegs))
        {
          if (   (inst->uiWriteAddr + inst->uiWriteQty)
              <= (*(mbs->pData)).stUnit[u].uiNbrHoldingRegs)
          {
            for (i = 0; i < inst->uiWriteQty; i++)
            {
              hreg = inst->uiWriteAddr + i;
              (*(mbs->pData)).stUnit[u].pHoldingRegs[hreg] = pHRegVal[(i)];
            }
          }
        }
      /*****************read multiple register ***************/
     if ( inst->puiReadVal == NULL)
        { inst->uiStatus = mbtERR_DATA_ADDRESS; goto END; }
      pHRegVal = (tHREG*) inst->puiReadVal;
      i = inst->uiReadAddr;
      if (i > mbs->pData->stUnit[u].uiNbrHoldingRegs)
        { inst->uiStatus = mbtERR_DATA_ADDRESS; goto END; }
      if (    (inst->uiReadQty > 0)
           && (inst->uiReadQty <= (*(mbs->pData)).stUnit[u].uiNbrHoldingRegs))
        {
          if (    (inst->uiReadAddr + inst->uiReadQty)
               <= (*(mbs->pData)).stUnit[u].uiNbrHoldingRegs)
          {
            for (i = 0; i < inst->uiReadQty; i++)
            {
              hreg = inst->uiReadAddr + i;
              pHRegVal[(i)] = mbs->pData->stUnit[u].pHoldingRegs[hreg];
            }
          }
        }
      break;
    default:
      { inst->uiStatus = mbtERR_ILLEGAL_FUNCTION; goto END; }
    }
    inst->uiStatus = ERR_OK;
  }
END: ; /* do nothing */
  /*=========================================================================*/
} /* fMBTSRW */

/*****************************************************************************
 * END OF CODE
 *****************************************************************************/
/*
  Local Variables:
  c-file-style: bsd
  c-basic-offset: 2
  comment-column: 45
  End:
*/
```

#### fMBTSFill.c
```c
/*****************************************************************************
 * Copyright:    B&R Industrie-Automation AG
 *
 * Project:      Library MBTCP
 *
 * Target:       B&R-PCC
 *
 * AR-Version:   B 2.01
 *
 * AS-Version:   V 3.0.71.16.SP01
 *
 * Filename:     fMBTSFill.c
 *
 * Function:     module-description
 *
 * Dependencies: description of all dependencies
 *
 *****************************************************************************
 * History:
 *
 * Version | Date        | Author      | Description
 * --------------------------------------------------------------------------
 *    1.00 | 2008-sep-19 | H.Anderes    | creation
 *****************************************************************************/

/*****************************************************************************
 * includes
 *****************************************************************************/
/* ansi-c import */
/* system import */
/* user defined import */
#include "MBTCP.h"
#include "MBTSlave.h"

/*****************************************************************************
 * type definitions
 *****************************************************************************/

/*****************************************************************************
 * functions
 *****************************************************************************/
/*===========================================================================*/
void fMBTSFill(struct fMBTSFill* inst)
/*---------------------------------------------------------------------------
  Function:

  Initialize the slave's data units (coils and registers) with
  values. Coils and Discrete Inputs are initialized with 0, 1,
  0... Input registers are filled with 1000, 1001, 1002... Holding
  registers are initialized with 0, 1, 2...

  History:

  Version | Date        | Author      | Description
  --------------------------------------------------------------------------
     1.00 | 2008-sep-19 | H.Anderes    | creation
  ===========================================================================*/
  {
  /* _LOCAL */
  UINT u, i, imax;
  /* _DYNAMIC */
  tstMBT_SVars* mbs;
  /*=========================================================================*/
  /* check if nil pointer */
  if (inst == NULL || inst->udiIdent == 0)
    {
    inst->uiStatus = mbtERR_NULL_POINTER;
	goto END;
    }
  mbs = (tstMBT_SVars *) inst->udiIdent;

  if (inst->bEnable < TRUE)
  {
    inst->uiStatus = ERR_FUB_ENABLE_FALSE;
  }
  else
  {
    inst->uiStatus = ERR_FUB_BUSY;

    for (u = mbs->pData->uiOffsetUnits; u < (mbs->pData->uiNbrUnits + mbs->pData->uiOffsetUnits); u++)
    {
      imax = mbs->pData->stUnit[u].uiNbrCoils;
      for (i = 0; i < imax; i++) {
        mbs->pData->stUnit[u].pCoils[i] = 0;
        mbs->pData->stUnit[u].pCoils[i] = (tCOIL)(i & 0x0001);
      }
      imax = mbs->pData->stUnit[u].uiNbrDiscreteInputs;
      for (i = 0; i < imax; i++) {
        mbs->pData->stUnit[u].pDiscreteInputs[i] = 0;
        mbs->pData->stUnit[u].pDiscreteInputs[i] = (tDINP)(i & 0x0001);
      }
      imax = mbs->pData->stUnit[u].uiNbrInputRegs;
      for (i = 0; i < imax; i++) {
        mbs->pData->stUnit[u].pInputRegs[i] = (tIREG)(1000 + i);
      }
      imax = mbs->pData->stUnit[u].uiNbrHoldingRegs;
      for (i = 0; i < imax; i++) {
        mbs->pData->stUnit[u].pHoldingRegs[i] = (tHREG)(i);
      }
    }
    mbs->bEnable = TRUE;
    inst->uiStatus = ERR_OK;
  }
  END: ; /* do nothing */
  /*=========================================================================*/
  } /* fMBTSFill */

/*****************************************************************************
 * END OF CODE
 *****************************************************************************/
```

#### fMBTMOpen.c
```c
/*****************************************************************************
 * Copyright:    B&R Industrie-Automation AG
 *
 * Project:      Library MBTCP
 *
 * Target:       B&R-PCC
 *
 * AR-Version:   B 2.01
 *
 * AS-Version:   V 3.0.71.16.SP01
 *
 * Filename:     fMBTMOpen.c
 *
 * Function:     module-description
 *
 * Dependencies: description of all dependencies
 *
 *****************************************************************************
 * History:
 *
 * Version | Date        | Author      | Description
 * ---------------------------------------------------------------------------
 *    1.00 | 2008-Oct-01 | H.Anderes    | creation
 *****************************************************************************/

/*****************************************************************************
 * includes
 *****************************************************************************/
/* ansi-c import */
/* system import */
/* user defined import */
#include "MBTCP.h"
#include "MBTMaster.h"

/*****************************************************************************
 * type definitions
 *****************************************************************************/

/*****************************************************************************
 * functions
 *****************************************************************************/
/*==========================================================================*/
void fMBTMOpen(struct fMBTMOpen* inst)
/*---------------------------------------------------------------------------
  Function:

  Allocates memory and pre-configures Modbus TCP Master.
  fMBTMOpen() should be called in the INIT section of a task prior
  to fMBTMaster(). See also fMBTMClose() to close the master in the
  task's EXIT section. The master connects to the Modbus TCP slave
  available at the IP address provided by szSlvIPAddr.

  History:

  Version | Date        | Author      | Description
  ---------------------------------------------------------------------------
     1.00 | 2008-Oct-01 | H.Anderes    | creation
  ===========================================================================*/
  {
  /* _LOCAL */
  UINT astatus = 0;
  RTInfo_typ stRTInfo;
  UDINT udiCycleTime;

  /* _DYNAMIC */
  tstMBT_MVars *mbm;
  tstMBT_MData *pData;

  /*=========================================================================*/
  if (inst == NULL)
  {
    inst->uiStatus = mbtERR_NULL_POINTER;
    goto END;
  }
  if (inst->bEnable < TRUE)
  {
    inst->uiStatus = ERR_FUB_ENABLE_FALSE;
  }
  else
  {
    inst->uiStatus = ERR_FUB_BUSY;
    if (inst->szSlvIPAddr == NULL)
    {
      inst->uiStatus = mbtERR_IP_ADRESS;
      goto END;
    }

    astatus = TMP_alloc(sizeof(tstMBT_MVars), (void**)&mbm);
    if (astatus > 0) { inst->uiStatus = astatus; goto END; }
    memset(mbm, 0, sizeof(tstMBT_MVars));
    astatus = TMP_alloc(sizeof(tstMBT_MData), (void**)&pData);
    if (astatus > 0) { inst->uiStatus = astatus; goto END; }
    memset(pData, 0, sizeof(tstMBT_MData));
    mbm->pData = pData;

    stRTInfo.enable = TRUE;
    RTInfo(&stRTInfo);
    udiCycleTime = (UDINT)(stRTInfo.cycle_time / 1000);
    stRTInfo.enable = FALSE;
    /* call RTInfo() */
    RTInfo(&stRTInfo);

    if (inst->uiPort < 1)
    {
      inst->uiPort = MBT_SLAVE_PORT;
    }
    if (inst->uiRecvTimeout < 1)
    {
      inst->uiRecvTimeout = RECV_TIMEOUT_DFLT;
    }

    memmove(&(mbm->slvIPAddr),&(inst->szSlvIPAddr), IPADDR_L);
    mbm->uiPort 	      = inst->uiPort;
    mbm->udiCycleTime	 = udiCycleTime;
    mbm->uiRecvTimeout = inst->uiRecvTimeout;
    mbm->uiStep		      = INIT;

    inst->udiIdent = (UDINT) mbm;
    if (inst->uiStatus == ERR_FUB_BUSY)         /* alloc OK */
    {
      inst->uiStatus = ERR_OK;
    }
  }
  END: ; /* do nothing */
  /*=========================================================================*/
  } /* fMBTMOpen */

/*****************************************************************************
 * END OF CODE
 *****************************************************************************/
 /*
Local Variables:
c-file-style: bsd
c-basic-offset: 2
comment-column: 45
End:
 */
```

#### fMBTMaster.c
```c
/****************************************************************************
 * Copyright:    B&R Industrie-Automation AG
 *
 * Project:      Library MBTCP
 *
 * Target:       B&R-PCC
 *
 * AR-Version:   B 2.01
 *
 * AS-Version:   V 3.0.71.16.SP01
 *
 * Filename:     fMBTMaster.c
 *
 * Function:     module-description
 *
 * Dependencies: description of all dependencies
 *
 ****************************************************************************
 * History:
 *
 * Version | Date        | Author      | Description
 * --------------------------------------------------------------------------
 *    1.00 | 2008-Oct-03 | H.Anderes    | creation
 *****************************************************************************/

/*****************************************************************************
 * includes
 *****************************************************************************/
/* ansi-c import */
/* system import */
/* user defined import */
#include "MBTCP.h"
#include "MBTMaster.h"

/*****************************************************************************
 * type definitions
 *****************************************************************************/

/*****************************************************************************
 * functions
 *****************************************************************************/
/*===========================================================================*/
void fMBTMaster(struct fMBTMaster* inst)
/*---------------------------------------------------------------------------
  Function:

  Modbus/TCP master (client) function. fMBTMaster()
  should be called in the CYCLIC section of a task after being
  configured by fMBTMOpen(). The master is closed by fMBTMClose().
  This master writes to or reads from a slave running fMBTSlave() or
  other widely available Modbus over TCP slave programs.

  History:

  Version | Date        | Author      | Description
  --------------------------------------------------------------------------
  1.00    | 2008-Oct-03 | H.Anderes    | creation
  ===========================================================================*/
{
  /* _LOCAL */
  /* _DYNAMIC */
  tstMBT_MVars *mbm;
  /*=========================================================================*/
  if (inst == NULL)
  {
    inst->uiStatus = mbtERR_NULL_POINTER;
    goto END;
  }
  mbm = (tstMBT_MVars *) inst->udiIdent;

  if (inst->bEnable < TRUE)
  {
    inst->uiStatus = ERR_FUB_ENABLE_FALSE;
  }
  else
  {

    mbm->bEnable = inst->bEnable;
    /* call fMBTMStates */
    fMBTMStates(mbm);

    inst->uiStep        = mbm->uiStep;
    inst->uiTxID        = mbm->uiTxID;
    inst->usiMBFuncCode = mbm->usiRecvBuf[7];
    inst->usiRxByteCnt  = mbm->usiRecvBuf[8];
	   strcpy(inst->szMsg,mbm->szMsg);
    inst->uiStatus      = mbm->uiStatus;
}

END: ; /* do nothing */
  /*=========================================================================*/
} /* fMBTMaster */

/*****************************************************************************
 * END OF CODE
 *****************************************************************************/
/*
  Local Variables:
  c-file-style: bsd
  c-basic-offset: 2
  comment-column: 45
  End:
 */
```

#### fMBTMClose.c
```c
/****************************************************************************
 * Copyright:    B&R Industrie-Automation AG
 *
 * Project:      Library MBTCP
 *
 * Target:       B&R-PCC
 *
 * AR-Version:   B 2.01
 *
 * AS-Version:   V 3.0.71.16.SP01
 *
 * Filename:     fMBTMClose.c
 *
 * Function:     module-description
 *
 * Dependencies: description of all dependencies
 *
 ****************************************************************************
 * History:
 *
 * Version | Date        | Author      | Description
 * --------------------------------------------------------------------------
 *    1.00 | 2008-Oct-03 | H.Anderes    | creation
 *****************************************************************************/

/*****************************************************************************
 * includes
 *****************************************************************************/
/* ansi-c import */
/* system import */
/* user defined import */
#include "MBTCP.h"
#include "MBTMaster.h"

/*****************************************************************************
 * type definitions
 *****************************************************************************/

/*****************************************************************************
 * functions
 *****************************************************************************/
/*===========================================================================*/
void fMBTMClose(struct fMBTMClose* inst)
/*---------------------------------------------------------------------------
  Function:

  Terminates a Modbus/TCP master (client) and releases allocated memory.
  fMBTMClose() should be called in the EXIT section of a task.
  See also fMBTMOpen() and fMBTMaster().

  History:

  Version | Date        | Author      | Description
  --------------------------------------------------------------------------
  1.00 | 2008-Oct-03 | H.Anderes    | creation
  5.00 | 2021-may-07 | W.Froehlich  | set correct FUB state fMBTMClose.uiStatus from ERR_FUB_BUSY to ERR_OK
  ===========================================================================*/
{
  /* _LOCAL */
  UINT fstatus = 0;
  USINT i;
  /* _DYNAMIC */
  tstMBT_MVars *mbm;
  /*=========================================================================*/
  if (inst == NULL)
  {
    inst->uiStatus = mbtERR_NULL_POINTER;
    goto END;
  }
  mbm = (tstMBT_MVars *) inst->udiIdent;

  if (inst->bEnable < TRUE)
  {
    inst->uiStatus = ERR_FUB_ENABLE_FALSE;
  }
  else
  {
		/* set correct FUB state fMBTSClose.uiStatus from ERR_FUB_BUSY to ERR_OK */
    inst->uiStatus = ERR_OK;

    /* disconnect from slave */
    mbm->uiStep = CLOSE_PORT;
    for (i = 0; i < 2; i++)                  /* 2 iterations needed */
      fMBTMStates(mbm);

    fstatus = TMP_free(sizeof(tstMBT_MData), (void**)mbm->pData);
    if (fstatus > 0)
    {
      inst->uiStatus = fstatus;
      ERRxwarning(fstatus, 0, (STRING*)"fMBTMClose: failed to TMP_free pData");
        goto END;
    }
    fstatus = TMP_free(sizeof(tstMBT_MVars), (void**)mbm);
    if (fstatus > 0)
    {
      inst->uiStatus = fstatus;
      ERRxwarning(fstatus, 0, (STRING*)"fMBTMClose: failed to TMP_free mbm");
      goto END;
    }
  }

END: ; /* do nothing */
  /*=========================================================================*/
} /* fMBTMClose */

/*****************************************************************************
 * END OF CODE
 *****************************************************************************/

/*
  Local Variables:
  c-file-style: bsd
  c-basic-offset: 2
  comment-column: 45
  End:
*/
```

#### fMBTMRW.c
```c
/*****************************************************************************
 * Copyright:    B&R Industrie-Automation AG
 *
 * Project:      Library MBTCP
 *
 * Target:       B&R-PCC
 *
 * AR-Version:   B 2.01
 *
 * AS-Version:   V 3.0.71.16.SP01
 *
 * Filename:     fMBTMRW.c
 *
 * Function:     module-description
 *
 * Dependencies: description of all dependencies
 *
 *****************************************************************************
 * History:
 *
 * Version | Date        | Author      | Description
 * --------------------------------------------------------------------------
 *    1.00 | 2008-Oct-03 | H.Anderes    | creation
 *****************************************************************************/

/*****************************************************************************
 * includes
 *****************************************************************************/
/* ansi-c import */
/* system import */
/* user defined import */
#include "MBTCP.h"
#include "MBTMaster.h"

/*****************************************************************************
 * type definitions
 *****************************************************************************/

/*****************************************************************************
 * functions
 *****************************************************************************/
/*===========================================================================*/
void fMBTMRW(struct fMBTMRW* inst)
/*---------------------------------------------------------------------------
  Function:

  Read/write individual values from/to coils and registers of given unit.
  The function code to use in member uiFcode of the passed structure is the
  same as for Modbus (0x01..0x06).

  History:

  Version | Date        | Author      | Description
  --------------------------------------------------------------------------
  1.00 | 2008-Oct-06 | H.Anderes    | creation
  ===========================================================================*/
{
  /* _LOCAL */
  /* _DYNAMIC */
  tstMBT_MVars* mbm;
  /*=========================================================================*/
  /* check if nil pointer */
  if (inst == NULL)
  {
    inst->uiStatus = mbtERR_NULL_POINTER;
	goto END;
  }
  mbm = (tstMBT_MVars *) inst->udiIdent;

  if (inst->bEnable < TRUE)
  {
    inst->uiStatus = ERR_FUB_ENABLE_FALSE;
  }
  else
  {
    inst->uiStatus = ERR_FUB_BUSY;

    mbm->pData->actParam[0].usiFCode	  = inst->usiFCode;
    mbm->pData->actParam[0].usiUnit 	  = inst->usiUnit;
    mbm->pData->actParam[0].uiReadAddr  = inst->uiReadAddr;
    mbm->pData->actParam[0].uiReadQty 	= inst->uiReadQty;
    mbm->pData->actParam[0].uiWriteAddr = inst->uiWriteAddr;
    mbm->pData->actParam[0].uiWriteQty  = inst->uiWriteQty;

    if (inst->bPoll)
    {
      mbm->pData->actEnable[0].bCyclic 	= TRUE;
      mbm->pData->actEnable[0].bSingle 	= FALSE;
      mbm->pData->actParam[0].udiTimer 	= inst->udiPollPeriod;
    }
    else
    {
      mbm->pData->actEnable[0].bCyclic 	= FALSE;
      mbm->pData->actEnable[0].bSingle 	= TRUE;
      mbm->pData->actParam[0].udiTimer 	= 0;
    }

    switch(inst->usiFCode)
    {
    case MBT_READ_COILS:                     /* 0x01 */
    case MBT_READ_DISCRETE_INPUTS:           /* 0x02 */
       if (inst->uiReadQty > MAX_COILS)
         { inst->uiStatus = mbtERR_MAX_NBR_COILS; inst->bRecvOK = FALSE; goto END; }
      break;
    case MBT_READ_HOLDING_REGISTERS:         /* 0x03 */
    case MBT_READ_INPUT_REGISTERS:           /* 0x04 */
      if (inst->uiReadQty > MAX_REGISTER) //same value as Holding register
         { inst->uiStatus = mbtERR_MAX_NBR_REGISTER; inst->bRecvOK = FALSE; goto END; }
      break;
    case MBT_WRITE_SINGLE_COIL:              /* 0x05 */
    case MBT_WRITE_MULTIPLE_COILS:           /* 0x0F */
     if (inst->uiWriteQty > MAX_COILS)
         { inst->uiStatus = mbtERR_MAX_NBR_COILS; inst->bRecvOK = FALSE; goto END; }
      break;
    case MBT_WRITE_SINGLE_REGISTER:          /* 0x06 */
    case MBT_WRITE_MULTIPLE_REGISTERS:       /* 0x10 */
      if (inst->uiWriteQty > MAX_REGISTER)
        { inst->uiStatus = mbtERR_MAX_NBR_REGISTER; inst->bRecvOK = FALSE; goto END; }
      break;
    case MBT_READ_WRITE_MULTIPLE_REGISTER:  /* 0x17 */
      if (    (inst->uiWriteQty > MAX_REGISTER)
           || (inst->uiReadQty > MAX_REGISTER))
        { inst->uiStatus = mbtERR_MAX_NBR_REGISTER; inst->bRecvOK = FALSE; goto END; }
      break;
    default:
      { inst->uiStatus = mbtERR_ILLEGAL_FUNCTION; goto END; }
    }

    switch(inst->usiFCode)
    {
    case MBT_READ_COILS:                     /* 0x01 */
    case MBT_READ_DISCRETE_INPUTS:           /* 0x02 */
    case MBT_READ_HOLDING_REGISTERS:         /* 0x03 */
    case MBT_READ_INPUT_REGISTERS:           /* 0x04 */
      if(inst->puiReadVal == NULL)
        { inst->uiStatus = mbtERR_DATA_ADDRESS; goto END; }
      mbm->pData->actParam[0].puiReadVal = (UDINT) inst->puiReadVal;
      break;
    case MBT_WRITE_SINGLE_COIL:              /* 0x05 */
    case MBT_WRITE_MULTIPLE_COILS:           /* 0x0F */
    case MBT_WRITE_SINGLE_REGISTER:          /* 0x06 */
    case MBT_WRITE_MULTIPLE_REGISTERS:       /* 0x10 */
      if( inst->puiWriteVal == NULL)
        { inst->uiStatus = mbtERR_DATA_ADDRESS; goto END; }
      mbm->pData->actParam[0].puiWriteVal = (UDINT) inst->puiWriteVal;
      break;
    case MBT_READ_WRITE_MULTIPLE_REGISTER:  /* 0x17 */
      if(    (inst->puiWriteVal == NULL)
          || (inst->puiReadVal == NULL))
        { inst->uiStatus = mbtERR_DATA_ADDRESS; goto END; }
      mbm->pData->actParam[0].puiReadVal  = (UDINT) inst->puiReadVal;
      mbm->pData->actParam[0].puiWriteVal = (UDINT) inst->puiWriteVal;
      break;
    default:
      { inst->uiStatus = mbtERR_ILLEGAL_FUNCTION; goto END; }
    }

    inst->bRecvOK = mbm->bRecvOK;
    inst->uiStatus = ERR_OK;
  }
END: ; /* do nothing */
  /*=========================================================================*/
} /* fMBTMRW */

/*****************************************************************************
 * END OF CODE
 *****************************************************************************/
/*
  Local Variables:
  c-file-style: bsd
  c-basic-offset: 2
  comment-column: 45
  End:
*/
```

#### MBTSlave.h
```c
/*****************************************************************************
 * Copyright:    B&R Industrie-Automation AG
 *
 * Project:      Library MBTCP
 *
 * Target:       B&R-PCC
 *
 * AR-Version:   B 2.01
 *
 * AS-Version:   V 3.0.71.16.SP01
 *
 * Filename:     MBTSlave.h
 *
 * Function:     module-description
 *
 * Dependencies: description of all dependencies
 *
 *****************************************************************************
 * History:
 *
 * Version | Date        | Author      | Description
 * --------------------------------------------------------------------------
 *    1.00 | 2008-sep-19 | H.Anderes    | creation
 *****************************************************************************/

/*****************************************************************************
 * includes
 *****************************************************************************/
#ifndef MBTSLAVE_H_
#define MBTSLAVE_H_

/* ansi-c import */
#include <string.h>
/* system import */
#include <bur/plc.h>                         /* IEC data types */
#include <asstring.h>
#include <astcp.h>
#include <convert.h>
#include <sys_lib.h>
#include <standard.h>                        /* used for POF() timer */
/* user defined import */
#include "MBTCP.h"

/*#define _MBTCP_LOGGER_DEBUG*/ /* if defined, errors are logged into the logger */
/*#define _MBTCP_LOGGER_EVENT*/ /* if defined, events are logged into the logger */

#ifdef __i386__
#define SWAPUINT        swapUINT
#define SWAPINT         swapINT
#define BYTE_OFFSET     0
#else
#define SWAPUINT
#define SWAPINT
#define BYTE_OFFSET     1
#endif

/*****************************************************************************
 * constants / macros
 *****************************************************************************/
#define NELEMS(array)           (sizeof(array) / sizeof(array[0]))
#define FALSE           0
#define TRUE            1

/* length of the request */
#define REQ_LEN_READ_COILS                      6
#define REQ_LEN_READ_DISCRETE_INPUTS            6
#define REQ_LEN_READ_HOLDING_REGISTERS          6
#define REQ_LEN_READ_INPUT_REGISTERS            6
#define REQ_LEN_WRITE_SINGLE_COIL               6
#define REQ_LEN_WRITE_SINGLE_REGISTER           6
#define REQ_LEN_WRITE_MULTIPLE_COILS            7
#define REQ_LEN_WRITE_MULTIPLE_REGISTERS        7
#define REQ_LEN_READ_WRITE_MULTIPLE_REGISTERS   11

#define MAX_COILS            2000
#define MAX_DISCRETE_INPUTS  2000
#define MAX_HOLDING_REGISTER 127
#define MAX_INPUT_REGISTER   127
/*****************************************************************************
 * type definitions
 *****************************************************************************/
/*
 * STEP values
 */
enum {
  MBCONF                = 1,
  INIT                  = 5,
  DISABLE               = 65534,
  OPEN_PORT             = 10,
  IOCTL                 = 15,
  WAIT_REQUEST          = 30,
  IOCTL_CLIENT          = 35,
  CLOSE_SLAVE           = 111,
  FATAL_ERROR0          = 240,
  FATAL_ERROR1          = 241,
  FATAL_ERROR2          = 242,
  FATAL_ERROR3          = 243,
  FATAL_ERROR4          = 244,
  FATAL_ERROR5          = 245,
  FATAL_ERROR6          = 246,
  FATAL_ERROR7          = 247,
  FATAL_ERROR8          = 248,
  FINAL_ERROR			        = 249
};

/*
 * Client Handler STEP values
 */
enum {
  enMBTCP_CLT_HANDLER_W4_REQUEST      = 0,
  enMBTCP_CLT_HANDLER_SEND_RESPONSE   = 1,
  enMBTCP_CLT_HANDLER_DISCONNECT      = 2
};

/* Booleans, switches
 */
enum {
  EXIT_FAILURE          = 1,
  ON                    = 0xFF00,
  OFF                   = 0x0000
};

/* Dimensions
 */
enum {
  MBT_SLAVE_PORT        = 502,
  MAX_OPEN_RETRIES      = 3,
  MBT_MAX_UNITS         = 300,
  NUNITS_DEF            = 1,             /* default num of Modbus units */
  OFFSET_NUNITS_DEF		   = 0,             /* default offset of Modnus units */
  MAX_CLIENT_REQUEST    = 5,
  MAX_CLIENT            = 5,
  MAX_CLOSE_LOOPS       = 1000,
  TIMEOUT_MS            = 1500,          /* receive TOF delay, in ms */
  MAX_RECV_BUFFER_LEN   = 1500,          /* was 128, max protocol = 260 bytes * 5 (Requests)*/
  MAX_SEND_BUFFER_LEN   = 300,           /* was 128, max protocol = 260 bytes */
  IPADDR_L              = 18,
  MESS_LEN              = 100,           /* error message length */
  HEADER_LEN            = 6,             /* Modbus header (MBAP) length */
  MIN_FRAME_LEN         = HEADER_LEN + 2 /* see analyze_req_from_client() */
};
/* MIN_FRAME_LEN =
   6 bytes for HEADER_LEN, Modbus Application Protocol (MBAP) header:
     bytes 0,1: transaction ID, incremented by client at every request
     bytes 2,3: protocol ID: 0x00 00 for ModbusTCP
     bytes 4,5: number of bytes in message to follow (0 to 252 bytes)
   1 byte:  server/slave unit ID (compulsory value)
   1 byte:  function code as defined in Modbus standard
   See also: http://www.scorpioncontrols.com/info/modbustcp.htm
             http://www.simplymodbus.ca/TCP.htm
             http://www.digitalbond.com/wiki/index.php/Modbus_TCP
             Page 5 of Modbus Application Protocol spec. V1.1b
*/

/* Modbus function codes
 */
enum {
  READ_COILS                            = 0x01,
  READ_DISCRETE_INPUTS                  = 0x02,
  READ_HOLDING_REGISTERS                = 0x03,
  READ_INPUT_REGISTERS                  = 0x04,
  WRITE_SINGLE_COIL                     = 0x05,
  WRITE_SINGLE_REGISTER                 = 0x06,
  WRITE_MULTIPLE_COILS                  = 0x0F,
  WRITE_MULTIPLE_REGISTERS              = 0x10,
  READ_WRITE_MULTIPLE_REGISTERS         = 0x17
};

/* Modbus protocol exception codes
 */
enum {
  MB_ILLEGAL_FUNCTION                   = 0x01,
  MB_ILLEGAL_DATA_ADDRESS               = 0x02,
  MB_ILLEGAL_DATA_VALUE                 = 0x03,
  MB_SLAVE_DEVICE_FAILURE               = 0x04,
  MB_ACKNOWLEDGE                        = 0x05,
  MB_SLAVE_DEVICE_BUSY                  = 0x06,
  MB_MEMORY_PARITY_ERROR                = 0x08,
  MB_GATEWAY_PATH_UNAVAILABLE           = 0x0A,
  MB_GATEWAY_TARGET_DEV_FAILED_RESPOND  = 0x0B
};

enum {
  mbtERR_NUM_BASE       = 50000 /* Modbus exceptions get added to this value */
};

typedef struct
{
  UINT  uiTxID;
  UINT  uiProtocolID;
  UINT  length;
  USINT usiUnit;
  USINT usiFCode;
} t_client_request;

typedef struct
{
  UINT  uiAddr;              /* starting address */
  UINT  uiQty;               /* quantity of coils, registers, etc. */
} t_read_request;

typedef struct
{
  UINT  uiAddr;              /* starting address */
  UINT  uiVal;
} t_single_write_request;

typedef struct
{
  UINT  uiAddr;
  UINT  uiQty;
  USINT usiByteNr;
} t_multiple_write_request;

typedef struct
{
  UINT  uiReadAddr;
  UINT  uiReadQty;
  UINT  uiWriteAddr;
  UINT  uiWriteQty;
  USINT usiByteNr;
} t_multiple_read_write_request;

typedef BOOL tCOIL;
typedef BOOL tDINP;
typedef UINT tIREG;
typedef UINT tHREG;

typedef struct
{
  UINT uiNbrCoils;
  UINT uiNbrDiscreteInputs;
  UINT uiNbrInputRegs;
  UINT uiNbrHoldingRegs;
  BOOL bCoilsExtern;
  BOOL bDiscreteInputsExtern;
  BOOL bInputRegsExtern;
  BOOL bHoldingRegsExtern;
  tCOIL *pCoils;
  tDINP *pDiscreteInputs;
  tIREG *pInputRegs;
  tHREG *pHoldingRegs;
} tstMBT_SUnit;

typedef struct
{
  UINT uiNbrUnits;
  UINT uiOffsetUnits;
  tstMBT_SUnit stUnit[MBT_MAX_UNITS];
} tstMBT_SData;

 typedef struct recv_buff_typ
 {
   USINT byte[MAX_RECV_BUFFER_LEN];
 } recv_buff_typ;

 typedef struct send_buff_typ
 {
   USINT byte[MAX_SEND_BUFFER_LEN];
   UINT  uiTxID;
   UINT  uiSendByte;
   UINT  uiReqLength;
 } send_buff_typ;

typedef struct
{
  BOOL                 bEnable;
  tstMBT_SData*        pData;
  UINT                 uiStep;
  UINT                 uiReturnStep;
  USINT                usiCltNr;     /* how many clients connected */
  USINT                usiCltServed; /* client currently served */
  tstclient_info       cltInfo[MAX_CLIENT];
  USINT                cltAddr[IPADDR_L];
  UINT                 uiPort;
  TcpOpen_typ          stTcpOpen;
  TcpIoctl_typ         stTcpIoctl;
  TcpServer_typ        stTcpServer;
  TcpSend_typ          stTcpSend[MAX_CLIENT];
  TcpRecv_typ          stTcpRecv[MAX_CLIENT];
  TcpClose_typ         stTcpClose[MAX_CLIENT];
  TOF_typ              TOFRecv[MAX_CLIENT];
  send_buff_typ        stSendBuf[MAX_CLIENT][MAX_CLIENT_REQUEST];
  USINT                usiReqIdx[MAX_CLIENT_REQUEST];
  recv_buff_typ        stRecvBuf[MAX_CLIENT]; /* all request are received in one buffer */
  USINT                usiNbrReq;
  UINT                 uiStatus;
  STRING               szMsg[MESS_LEN];
  BOOL                 bClosing;
  tcpLINGER_typ        sLinger;
  UINT                 uiStepCltHandler[MAX_CLIENT];
  /*Additional Data*/
  USINT				            usiOpenRetries;
  UDINT				            udiRecvCnt;
  UDINT				            udiSendCnt;
  UINT				             uiOffsetUnits;
} tstMBT_SVars;

/*****************************************************************************
 * functions protoytpes
 ****************************************************************************/
UINT arr_alloc                    (UDINT size, UDINT* p_reg);
UINT fMBTSStates                  (tstMBT_SVars* inst);
UINT add_client                   (tstMBT_SVars* inst);
void remove_client                (tstMBT_SVars* inst, USINT client);
void recv_client                  (tstMBT_SVars* inst, UINT i);
void send_response                (tstMBT_SVars* inst, UINT i);
void disconnect_client            (tstMBT_SVars* inst, UINT i);
void client_handler               (tstMBT_SVars* inst);
UINT analyze_req_from_client      (tstMBT_SVars* inst, USINT client);
void create_exception_response    (tstMBT_SVars* inst, USINT client, USINT req, UINT reqOffset, USINT excode);
void read_discrete_inputs         (tstMBT_SVars* inst, USINT client, USINT req, UINT reqOffset);
void read_coils                   (tstMBT_SVars* inst, USINT client, USINT req, UINT reqOffset);
void read_holding_registers       (tstMBT_SVars* inst, USINT client, USINT req, UINT reqOffset);
void read_input_registers         (tstMBT_SVars* inst, USINT client, USINT req, UINT reqOffset);
void write_single_coil            (tstMBT_SVars* inst, USINT client, USINT req, UINT reqOffset);
void write_single_register        (tstMBT_SVars* inst, USINT client, USINT req, UINT reqOffset);
void write_multiple_coils         (tstMBT_SVars* inst, USINT client, USINT req, UINT reqOffset);
void write_multiple_registers     (tstMBT_SVars* inst, USINT client, USINT req, UINT reqOffset);
void read_write_multiple_registers(tstMBT_SVars* inst, USINT clt, USINT req, UINT reqOffset);
void mberror                      (tstMBT_SVars* inst);
void mberror_client               (tstMBT_SVars* inst, USINT clt);
void exit (void) __attribute__ ((__noreturn__));

/*****************************************************************************
 * END OF CODE
 *****************************************************************************/
/*
Local Variables:
c-file-style: bsd
c-basic-offset: 2
comment-column: 45
End:
 */
#endif /* MBTSLAVE_H_ */
```
